# EPICS substitutions: sandalsSampleChangerApp/Db/sandals_sample_changer_beckhoff_extras.substitutions
file "$(TOP)/beckhoffApp/beckhoff_read_pv.template" {
    pattern {P, NAME, PORT, ADSPORT, V, RECTYPE, EPICSDTYP, ADS_TYPE}
    {"\$(P)", "FPT100_04", "\$(PORT)", "\$(ADSPORT)", "Sample_Changer.fPt100_04", "ai", "asynFloat64", "LREAL"}
    {"\$(P)", "FPT100_10", "\$(PORT)", "\$(ADSPORT)", "Sample_Changer.fPt100_10", "ai", "asynFloat64", "LREAL"}
    {"\$(P)", "FPT100_14", "\$(PORT)", "\$(ADSPORT)", "Sample_Changer.fPt100_14", "ai", "asynFloat64", "LREAL"}
}
